// TwinCAT 3 PLC project Tests
// ProgramVersion: 3.1.4022.3
// libraries:
//   lcls-twincat-motion-zlentz, * (SLAC)
//   Tc2_Standard, * (Beckhoff Automation GmbH)
//   Tc2_System, * (Beckhoff Automation GmbH)
//   Tc3_Module, * (Beckhoff Automation GmbH)
// project tree:
//   / PlcTask.TcTTO
//   POUs/ MAIN.TcPOU
// real-time tasks:
//   TASK PlcTask: cycle T#10ms, priority 20, ADS port 350
// motion (NC):
//   TASK NC-Task 1 SAF: cycle T#2ms, priority 4, ADS port 501
//   TASK NC-Task 1 SVB: cycle T#10ms, priority 8, ADS port 511
//   AXIS Axis 1 (id 1)
//     OtherSettings: AllowMotionCmdToSlave=true
//     encoder EncType=1
//     drive DrvType=5
//       Analog: ScaleFactorActTorque=0.1
//     controller CtrType=1
//       CtrPara: PriorControlFactor=1
//         Observer: BandWidth=20
// variable links:
//   Library Instance <-> NC-Task 1 SAF/Axes/Axis_AtPositionState_Test
//     PlcTask Inputs/PRG_TEST.fb_AtPositionState_Test.stMotionStage.Axis.NcToPlc <-> Outputs/ToPlc
//     PlcTask Outputs/PRG_TEST.fb_AtPositionState_Test.stMotionStage.Axis.PlcToNc <-> Inputs/FromPlc
//   Library Instance <-> NC-Task 1 SAF/Axes/Axis_AxisParameter_Test
//     PlcTask Inputs/PRG_TEST.fb_AxisParameterSetExposed_Test.stMotionStage.Axis.NcToPlc <-> Outputs/ToPlc
//     PlcTask Outputs/PRG_TEST.fb_AxisParameterSetExposed_Test.stMotionStage.Axis.PlcToNc <-> Inputs/FromPlc
//   Library Instance <-> NC-Task 1 SAF/Axes/Axis_BacklashCompensation_Test
//     PlcTask Inputs/PRG_TEST.fb_MotionBacklashCompensation_Test.stMotionStage.Axis.NcToPlc <-> Outputs/ToPlc
//     PlcTask Outputs/PRG_TEST.fb_MotionBacklashCompensation_Test.stMotionStage.Axis.PlcToNc <-> Inputs/FromPlc
//   Library Instance <-> NC-Task 1 SAF/Axes/Axis_MotionVirtualFrameRx_Test
//     PlcTask Inputs/PRG_TEST.fbMotionVirtualFrameTest.stMotionStageRx.Axis.NcToPlc <-> Outputs/ToPlc
//     PlcTask Outputs/PRG_TEST.fbMotionVirtualFrameTest.stMotionStageRx.Axis.PlcToNc <-> Inputs/FromPlc
//   Library Instance <-> NC-Task 1 SAF/Axes/Axis_MotionVirtualFrameRy_Test
//     PlcTask Inputs/PRG_TEST.fbMotionVirtualFrameTest.stMotionStageRy.Axis.NcToPlc <-> Outputs/ToPlc
//     PlcTask Outputs/PRG_TEST.fbMotionVirtualFrameTest.stMotionStageRy.Axis.PlcToNc <-> Inputs/FromPlc
//   Library Instance <-> NC-Task 1 SAF/Axes/Axis_MotionVirtualFrameRz_Test
//     PlcTask Inputs/PRG_TEST.fbMotionVirtualFrameTest.stMotionStageRz.Axis.NcToPlc <-> Outputs/ToPlc
//     PlcTask Outputs/PRG_TEST.fbMotionVirtualFrameTest.stMotionStageRz.Axis.PlcToNc <-> Inputs/FromPlc
//   Library Instance <-> NC-Task 1 SAF/Axes/Axis_MotionVirtualFrameVx_Test
//     PlcTask Inputs/PRG_TEST.fbMotionVirtualFrameTest.stMotionStageVx.Axis.NcToPlc <-> Outputs/ToPlc
//     PlcTask Outputs/PRG_TEST.fbMotionVirtualFrameTest.nPositionCountsVx <-> Enc/Inputs/In/nDataIn1
//     PlcTask Outputs/PRG_TEST.fbMotionVirtualFrameTest.stMotionStageVx.Axis.PlcToNc <-> Inputs/FromPlc
//   Library Instance <-> NC-Task 1 SAF/Axes/Axis_MotionVirtualFrameVy_Test
//     PlcTask Inputs/PRG_TEST.fbMotionVirtualFrameTest.stMotionStageVy.Axis.NcToPlc <-> Outputs/ToPlc
//     PlcTask Outputs/PRG_TEST.fbMotionVirtualFrameTest.nPositionCountsVy <-> Enc/Inputs/In/nDataIn1
//     PlcTask Outputs/PRG_TEST.fbMotionVirtualFrameTest.stMotionStageVy.Axis.PlcToNc <-> Inputs/FromPlc
//   Library Instance <-> NC-Task 1 SAF/Axes/Axis_MotionVirtualFrameVz_Test
//     PlcTask Inputs/PRG_TEST.fbMotionVirtualFrameTest.stMotionStageVz.Axis.NcToPlc <-> Outputs/ToPlc
//     PlcTask Outputs/PRG_TEST.fbMotionVirtualFrameTest.nPositionCountsVz <-> Enc/Inputs/In/nDataIn1
//     PlcTask Outputs/PRG_TEST.fbMotionVirtualFrameTest.stMotionStageVz.Axis.PlcToNc <-> Inputs/FromPlc
//   Library Instance <-> NC-Task 1 SAF/Axes/Axis_NCErrorFFO_Test
//     PlcTask Inputs/PRG_TEST.fb_NCErrorFFO_Test.stMotionStage.Axis.NcToPlc <-> Outputs/ToPlc
//     PlcTask Outputs/PRG_TEST.fb_NCErrorFFO_Test.stMotionStage.Axis.PlcToNc <-> Inputs/FromPlc
//   Library Instance <-> NC-Task 1 SAF/Axes/Axis_PositionStateMoveND_Test_1
//     PlcTask Inputs/PRG_TEST.fb_PositionStateMoveND_Test.astMotionStage[1].Axis.NcToPlc <-> Outputs/ToPlc
//     PlcTask Outputs/PRG_TEST.fb_PositionStateMoveND_Test.astMotionStage[1].Axis.PlcToNc <-> Inputs/FromPlc
//   Library Instance <-> NC-Task 1 SAF/Axes/Axis_PositionStateMoveND_Test_2
//     PlcTask Inputs/PRG_TEST.fb_PositionStateMoveND_Test.astMotionStage[2].Axis.NcToPlc <-> Outputs/ToPlc
//     PlcTask Outputs/PRG_TEST.fb_PositionStateMoveND_Test.astMotionStage[2].Axis.PlcToNc <-> Inputs/FromPlc
//   Library Instance <-> NC-Task 1 SAF/Axes/Axis_PositionStateMoveND_Test_3
//     PlcTask Inputs/PRG_TEST.fb_PositionStateMoveND_Test.astMotionStage[3].Axis.NcToPlc <-> Outputs/ToPlc
//     PlcTask Outputs/PRG_TEST.fb_PositionStateMoveND_Test.astMotionStage[3].Axis.PlcToNc <-> Inputs/FromPlc
//   Library Instance <-> NC-Task 1 SAF/Axes/Axis_PositionStateMove_Test
//     PlcTask Inputs/PRG_TEST.fb_PositionStateMove_Test.stMotionStage.Axis.NcToPlc <-> Outputs/ToPlc
//     PlcTask Outputs/PRG_TEST.fb_PositionStateMove_Test.stMotionStage.Axis.PlcToNc <-> Inputs/FromPlc
//   Library Instance <-> NC-Task 1 SAF/Axes/Axis_PositionStateND_Test_1
//     PlcTask Inputs/PRG_TEST.fb_PositionStateND_Test.stMotionStage1.Axis.NcToPlc <-> Outputs/ToPlc
//     PlcTask Outputs/PRG_TEST.fb_PositionStateND_Test.stMotionStage1.Axis.PlcToNc <-> Inputs/FromPlc
//   Library Instance <-> NC-Task 1 SAF/Axes/Axis_PositionStateND_Test_2
//     PlcTask Inputs/PRG_TEST.fb_PositionStateND_Test.stMotionStage2.Axis.NcToPlc <-> Outputs/ToPlc
//     PlcTask Outputs/PRG_TEST.fb_PositionStateND_Test.stMotionStage2.Axis.PlcToNc <-> Inputs/FromPlc
//   Library Instance <-> NC-Task 1 SAF/Axes/Axis_PositionStateND_Test_3
//     PlcTask Inputs/PRG_TEST.fb_PositionStateND_Test.stMotionStage3.Axis.NcToPlc <-> Outputs/ToPlc
//     PlcTask Outputs/PRG_TEST.fb_PositionStateND_Test.stMotionStage3.Axis.PlcToNc <-> Inputs/FromPlc
//   Library Instance <-> NC-Task 1 SAF/Axes/Axis_PositionStatePMPSND_Test_1
//     PlcTask Inputs/PRG_TEST.fb_PositionStatePMPSND_Test.stMotionStage1.Axis.NcToPlc <-> Outputs/ToPlc
//     PlcTask Outputs/PRG_TEST.fb_PositionStatePMPSND_Test.stMotionStage1.Axis.PlcToNc <-> Inputs/FromPlc
//   Library Instance <-> NC-Task 1 SAF/Axes/Axis_PositionStatePMPSND_Test_2
//     PlcTask Inputs/PRG_TEST.fb_PositionStatePMPSND_Test.stMotionStage2.Axis.NcToPlc <-> Outputs/ToPlc
//     PlcTask Outputs/PRG_TEST.fb_PositionStatePMPSND_Test.stMotionStage2.Axis.PlcToNc <-> Inputs/FromPlc
//   Library Instance <-> NC-Task 1 SAF/Axes/Axis_PositionStatePMPSND_Test_3
//     PlcTask Inputs/PRG_TEST.fb_PositionStatePMPSND_Test.stMotionStage3.Axis.NcToPlc <-> Outputs/ToPlc
//     PlcTask Outputs/PRG_TEST.fb_PositionStatePMPSND_Test.stMotionStage3.Axis.PlcToNc <-> Inputs/FromPlc
//   Library Instance <-> NC-Task 1 SAF/Axes/Axis_PositionStateReadND_Test_1
//     PlcTask Inputs/PRG_TEST.fb_PositionStateReadND_Test.astMotionStage[1].Axis.NcToPlc <-> Outputs/ToPlc
//     PlcTask Outputs/PRG_TEST.fb_PositionStateReadND_Test.astMotionStage[1].Axis.PlcToNc <-> Inputs/FromPlc
//   Library Instance <-> NC-Task 1 SAF/Axes/Axis_PositionStateReadND_Test_2
//     PlcTask Inputs/PRG_TEST.fb_PositionStateReadND_Test.astMotionStage[2].Axis.NcToPlc <-> Outputs/ToPlc
//     PlcTask Outputs/PRG_TEST.fb_PositionStateReadND_Test.astMotionStage[2].Axis.PlcToNc <-> Inputs/FromPlc
//   Library Instance <-> NC-Task 1 SAF/Axes/Axis_PositionStateReadND_Test_3
//     PlcTask Inputs/PRG_TEST.fb_PositionStateReadND_Test.astMotionStage[3].Axis.NcToPlc <-> Outputs/ToPlc
//     PlcTask Outputs/PRG_TEST.fb_PositionStateReadND_Test.astMotionStage[3].Axis.PlcToNc <-> Inputs/FromPlc
//   Library Instance <-> NC-Task 1 SAF/Axes/Axis_PositionStateReadND_Test_4
//     PlcTask Inputs/PRG_TEST.fb_PositionStateReadND_Test.astSqMotionStage[1].Axis.NcToPlc <-> Outputs/ToPlc
//     PlcTask Outputs/PRG_TEST.fb_PositionStateReadND_Test.astSqMotionStage[1].Axis.PlcToNc <-> Inputs/FromPlc
//   Library Instance <-> NC-Task 1 SAF/Axes/Axis_PositionStateReadND_Test_5
//     PlcTask Inputs/PRG_TEST.fb_PositionStateReadND_Test.astSqMotionStage[2].Axis.NcToPlc <-> Outputs/ToPlc
//     PlcTask Outputs/PRG_TEST.fb_PositionStateReadND_Test.astSqMotionStage[2].Axis.PlcToNc <-> Inputs/FromPlc
//   Library Instance <-> NC-Task 1 SAF/Axes/Axis_PositionStateRead_Test
//     PlcTask Inputs/PRG_TEST.fb_PositionStateRead_Test.stMotionStage.Axis.NcToPlc <-> Outputs/ToPlc
//     PlcTask Outputs/PRG_TEST.fb_PositionStateRead_Test.stMotionStage.Axis.PlcToNc <-> Inputs/FromPlc
//   Library Instance <-> NC-Task 1 SAF/Axes/Axis_PowerEnableMode_Test
//     PlcTask Inputs/PRG_TEST.fb_PowerEnableMode_Test.stMotionStage.Axis.NcToPlc <-> Outputs/ToPlc
//     PlcTask Outputs/PRG_TEST.fb_PowerEnableMode_Test.stMotionStage.Axis.PlcToNc <-> Inputs/FromPlc
//   Library Instance <-> NC-Task 1 SAF/Axes/Axis_StatePMPSEnable_Test
//     PlcTask Inputs/PRG_TEST.fb_StatePMPSEnables_Test.stMotionStage.Axis.NcToPlc <-> Outputs/ToPlc
//     PlcTask Outputs/PRG_TEST.fb_StatePMPSEnables_Test.stMotionStage.Axis.PlcToNc <-> Inputs/FromPlc
//   Library Instance <-> NC-Task 1 SAF/Axes/Axis_TestHelperSetAndMove_Test
//     PlcTask Inputs/PRG_TEST.fb_TestHelperSetAndMove_Test.stMotionStage.Axis.NcToPlc <-> Outputs/ToPlc
//     PlcTask Outputs/PRG_TEST.fb_TestHelperSetAndMove_Test.stMotionStage.Axis.PlcToNc <-> Inputs/FromPlc
//   Library Instance <-> NC-Task 1 SAF/Axes/Axis_TestStateInitTiming
//     PlcTask Inputs/PRG_TEST.fb_TestStateInitTiming.stMotionStage.Axis.NcToPlc <-> Outputs/ToPlc
//     PlcTask Outputs/PRG_TEST.fb_TestStateInitTiming.stMotionStage.Axis.PlcToNc <-> Inputs/FromPlc

CONFIGURATION Tests
    RESOURCE PLC ON TwinCAT3
        TASK PlcTask(INTERVAL := T#10ms, PRIORITY := 20);
        PROGRAM MAIN WITH PlcTask : MAIN;
    END_RESOURCE
END_CONFIGURATION

// ---- POUs/MAIN.TcPOU
PROGRAM MAIN
VAR
	M1: DUT_MotionStage;
	fbMotionStage: FB_MotionStage;
	nCounter: UINT;
END_VAR

fbMotionStage(stMotionStage:=M1);
nCounter := nCounter + 1;

END_PROGRAM
